INTERFACE ITF_LTU EXTENDS ITF_Device

PROPERTY CarrierPresent : BOOL
GET
END_GET
SET
END_SET
END_PROPERTY

PROPERTY LTUFree : BOOL
GET
END_GET
SET
END_SET
END_PROPERTY

PROPERTY LTUPosition : E_LTUPosition
GET
END_GET
SET
END_SET
END_PROPERTY

METHOD mCmdExec_MoveMiddle : E_CmdState
VAR_INPUT
	I_bExecute					: BOOL;
END_VAR
END_METHOD

METHOD mCmdExec_MoveTop : E_CmdState
VAR_INPUT
	I_bExecute					: BOOL;
END_VAR
END_METHOD

METHOD mCmdExec_TransferTop : E_CmdState
VAR_INPUT
	I_bExecute					: BOOL;
END_VAR
END_METHOD

METHOD mGetLTUByConvoyer : E_CmdState
VAR_INPUT
	I_bExecute					: BOOL;
END_VAR
END_METHOD

PROPERTY ReservedBy : E_Convoyer
GET
END_GET
SET
END_SET
END_PROPERTY

END_INTERFACE

(* stored: Version 1.1.0.1, ProductVersion 3.1.4026.18
   Itf ITF_LTU: Id {6c0d6849-e396-4313-9db5-4e08f7814412}
   Folder 01 Properties: Id {918ca8a6-e0b0-4e1d-9c02-fec848137e0f}
   Folder 02 Methodes: Id {52451a06-1a21-4dc8-86d8-33d6b2f2007a}
   Property CarrierPresent: Id {3edd6f5f-6da5-4acc-96c1-1a9245c92eb7}
   Get Get: Id {42de535c-13e8-4f5f-8400-33ca1492df76}
   Set Set: Id {26b3fc33-8256-408e-8a8d-b46d2057804b}
   Property LTUFree: Id {3c50412d-7b7a-4f29-b7b2-a28bde9f6fe5}
   Get Get: Id {4f194186-e093-4e45-aaa1-47844022f82b}
   Set Set: Id {11087894-221b-4eee-b108-75a26939d905}
   Property LTUPosition: Id {4e70c088-9f39-4b77-87a2-e5e8c87d9ec5}
   Get Get: Id {52a9326c-be79-41ea-920c-a613d38c0be4}
   Set Set: Id {925464df-cff8-4827-b5d7-bc532a493b28}
   Method mCmdExec_MoveMiddle: Id {065f028c-a162-4f8e-ad8f-163ada6683f3}
   Method mCmdExec_MoveTop: Id {dd172e8b-57a6-4c50-aedb-1b42c50c4b0f}
   Method mCmdExec_TransferTop: Id {0699606b-20d9-450f-ac58-6e4a863820c1}
   Method mGetLTUByConvoyer: Id {9ddedb5f-5861-4538-808c-36f0d32352cb}
   Property ReservedBy: Id {3282ed56-d078-4912-b714-d61a45b4bf20}
   Get Get: Id {b869b8e0-48e0-42f6-990b-b68194ec4278}
   Set Set: Id {8f605f2e-5c6b-4860-b6d8-424710527a42} *)
